// TwinCAT 3 PLC project TcAbbLinkin
// Title: TcAbbLinkin
// Company: Loupe
// Author: Loupe
// ProjectVersion: 0.1.0
// ProgramVersion: 3.1.4024.0
// libraries:
//   Tc2_Standard, * (Beckhoff Automation GmbH)
//   Tc2_System, * (Beckhoff Automation GmbH)
//   Tc2_Utilities, * (Beckhoff Automation GmbH)
//   Tc3_IotBase, * (Beckhoff Automation GmbH)
//   Tc3_JsonXml, * (Beckhoff Automation GmbH)
//   Tc3_Module, * (Beckhoff Automation GmbH)
// project tree:
//   DUTs/ AbbLinkinAuthDigest_Typ.TcDUT (not stored), AbbLinkinConfiguration_Typ.TcDUT, AbbLinkinRequestResults_Typ.TcDUT, AbbLinkinRequest_Typ.TcDUT (not stored), AbbLinkinRequestQueue_Typ.TcDUT (not stored), AbbLinkinRequestStatus_Typ.TcDUT, AbbLinkinAuth_Typ.TcDUT (not stored), ABBLINKIN_AUTH_HEADER_VALUE.TcDUT, ABBLINKIN_RWS_API_VERSION.TcDUT, ABBLINKIN_STATE.TcDUT, ABBLINKIN_COMMAND_TYPE.TcDUT, ABBLINKIN_DATA_TYPE_Typ.TcDUT (not stored), ABBLINKIN_STRING_EX_LEN.TcDUT
//   / PlcTask.TcTTO (not stored)
//   POUs/ MAIN.TcPOU, Example.TcPOU, TcAbbLinkin.TcPOU (not stored)
// real-time tasks:
//   TASK PlcTask: cycle T#10ms, priority 20, ADS port 350

// ---- DUTs/AbbLinkinConfiguration_Typ.TcDUT
// Copyright (c) 2024 Loupe (https://loupe.team), provided under the MIT License.
TYPE AbbLinkinConfiguration_Typ :
STRUCT
	rwsIpAddress : STRING := '127.0.0.1';
	rwsTcpPort : USINT := 80;
	rwsVersion : ABBLINKIN_RWS_API_VERSION;
	rwsUsername : STRING := 'Default User';
	rwsPassword : STRING := 'robotics';
	tlsAllowRwsCertSelfSigned : BOOL := FALSE;
	tlsCAFile : STRING(255) := '';
END_STRUCT
END_TYPE

// ---- DUTs/AbbLinkinRequestResults_Typ.TcDUT
// Copyright (c) 2024 Loupe (https://loupe.team), provided under the MIT License.
TYPE AbbLinkinRequestResults_Typ :
STRUCT
	pDataBool : POINTER TO BOOL;
	pDataDint : POINTER TO DINT;
	pDataLreal : POINTER TO LREAL;
	pDataString : POINTER TO STRING;
	dataType : ABBLINKIN_DATA_TYPE_Typ;
	dataLen : INT;
END_STRUCT
END_TYPE

// ---- DUTs/AbbLinkinRequestStatus_Typ.TcDUT
// Copyright (c) 2024 Loupe (https://loupe.team), provided under the MIT License.
TYPE AbbLinkinRequestStatus_Typ :
STRUCT
	busy : BOOL;
	done : BOOL;
	error : BOOL;
	errorID : DINT;
	errorMsg : STRING;
END_STRUCT
END_TYPE

// ---- DUTs/ABBLINKIN_AUTH_HEADER_VALUE.TcDUT
// Copyright (c) 2024 Loupe (https://loupe.team), provided under the MIT License.
{attribute 'qualified_only'}
{attribute 'strict'}
TYPE ABBLINKIN_AUTH_HEADER_VALUE :
(
	NONE,
	BASIC,
	DIGEST
);
END_TYPE

// ---- DUTs/ABBLINKIN_RWS_API_VERSION.TcDUT
// Copyright (c) 2024 Loupe (https://loupe.team), provided under the MIT License.
{attribute 'qualified_only'}
{attribute 'strict'}
TYPE ABBLINKIN_RWS_API_VERSION :
(
	V1 := 0,
	V2 := 2
);
END_TYPE

// ---- DUTs/ABBLINKIN_STATE.TcDUT
// Copyright (c) 2024 Loupe (https://loupe.team), provided under the MIT License.
{attribute 'qualified_only'}
{attribute 'strict'}
TYPE ABBLINKIN_STATE :
(
	IDLE,
	SEND_REQUEST,
	WAIT_FOR_RESONSE,
	PROCESS_RESPONSE,
	AUTH_START,
	AUTH_SEND_REQUEST,
	AUTH_WAIT_FOR_RESONSE,
	AUTH_PROCESS_RESPONSE,
	AUTH_DIGEST_RESPONSE_CALCULATE,
	AUTH_DIGEST_RESPONSE_SEND,
	ERROR
);
END_TYPE

// ---- DUTs/ABBLINKIN_COMMAND_TYPE.TcDUT
// Copyright (c) 2024 Loupe (https://loupe.team), provided under the MIT License.
{attribute 'qualified_only'}
{attribute 'strict'}
TYPE ABBLINKIN_COMMAND_TYPE :
(
	GET_IO,
	GET_CTRL_STATE,
	GET_OP_MODE,
	GET_RAPID_STATE,
	GET_SYMBOL,
	POWER_OFF,
	POWER_ON,
	RAPID_RESET,
	RAPID_START,
	RAPID_STOP,
	SET_IO,
	SET_SYMBOL
);
END_TYPE

// ---- DUTs/ABBLINKIN_STRING_EX_LEN.TcDUT
// Copyright (c) 2024 Loupe (https://loupe.team), provided under the MIT License.
TYPE ABBLINKIN_STRING_EX_LEN : STRING(2000); END_TYPE

// ---- POUs/MAIN.TcPOU
// Copyright (c) 2024 Loupe (https://loupe.team), provided under the MIT License.
PROGRAM MAIN
VAR
	myRobotLink : TcAbbLinkin;
	userSetConfigurationNow : BOOL := TRUE;
	userConnectStartNow : BOOL := TRUE;
	userConnectStopNow : BOOL;
	
	userGetCtrlStateNow : BOOL;
	userGetCtrlStateStatus : AbbLinkinRequestStatus_Typ;
	userGetCtrlStateResult : STRING;
	
	userGetOpModeNow : BOOL;
	userGetOpModeStatus : AbbLinkinRequestStatus_Typ;
	userGetOpModeResult : STRING;
	
	userGetRapidStateNow : BOOL;
	userGetRapidStateStatus : AbbLinkinRequestStatus_Typ;
	userGetRapidStateResult : STRING;
	
	userGetIoBoolNow : BOOL;
	userGetIoBoolStatus : AbbLinkinRequestStatus_Typ;
	userGetIoBoolResult : BOOL;
	
	userGetIoLrealNow : BOOL;
	userGetIoLrealStatus : AbbLinkinRequestStatus_Typ;
	userGetIoLrealResult : LREAL;
	
	userGetIoDintNow : BOOL;
	userGetIoDintStatus : AbbLinkinRequestStatus_Typ;
	userGetIoDintResult : DINT;
	
	
	userSetIoBoolNow : BOOL;
	userSetIoBoolValue : BOOL := 1;
	userSetIoBoolStatus : AbbLinkinRequestStatus_Typ;
	userSetIoDintNow : BOOL;
	userSetIoDintValue : DINT := 57;
	userSetIoDintStatus : AbbLinkinRequestStatus_Typ;
	userSetIoLrealNow : BOOL;
	userSetIoLrealValue : LREAL := 41.123456;
	userSetIoLrealStatus : AbbLinkinRequestStatus_Typ;
	
	
	userGetSymbolBoolNow : BOOL;
	userGetSymbolBoolResult : BOOL;
	userGetSymbolBoolStatus : AbbLinkinRequestStatus_Typ;
	userGetSymbolNumNow : BOOL;
	userGetSymbolNumResult : LREAL;
	userGetSymbolNumStatus : AbbLinkinRequestStatus_Typ;
	userGetSymbolStringNow : BOOL;
	userGetSymbolStringResult : STRING;
	userGetSymbolStringStatus : AbbLinkinRequestStatus_Typ;
	
	userSetSymbolBoolNow : BOOL;
	userSetSymbolBoolValue : BOOL := 1;
	userSetSymbolBoolStatus : AbbLinkinRequestStatus_Typ;
	userSetSymbolDintNow : BOOL;
	userSetSymbolDintValue : DINT := -57;
	userSetSymbolDintStatus : AbbLinkinRequestStatus_Typ;
	userSetSymbolLrealNow : BOOL;
	userSetSymbolLrealValue : LREAL := -41.123456;
	userSetSymbolLrealStatus : AbbLinkinRequestStatus_Typ;
	userSetSymbolStringNow : BOOL;
	userSetSymbolStringValue : STRING := 'test String';
	userSetSymbolStringStatus : AbbLinkinRequestStatus_Typ;
	userSetSymbolWStringNow : BOOL;
	userSetSymbolWStringValue : WSTRING := "test WString";
	userSetSymbolWStringStatus : AbbLinkinRequestStatus_Typ;
	
	
	userPowerOffNow : BOOL;
	userPowerOffStatus : AbbLinkinRequestStatus_Typ;
	userPowerOnNow : BOOL;
	userPowerOnStatus : AbbLinkinRequestStatus_Typ;
	userRapidResetNow : BOOL;
	userRapidResetStatus : AbbLinkinRequestStatus_Typ;
	userRapidStopNow : BOOL;
	userRapidStopStatus : AbbLinkinRequestStatus_Typ;
	userRapidStartNow : BOOL;
	userRapidStartStatus : AbbLinkinRequestStatus_Typ;
	
	
	userAckErrorNow : BOOL;
END_VAR

// Set configuration
if userSetConfigurationNow then
	myRobotLink.configuration.rwsIpAddress := '127.0.0.1';
	myRobotLink.configuration.rwsTcpPort := 80;
	myRobotLink.configuration.rwsVersion := ABBLINKIN_RWS_API_VERSION.V2;
	myRobotLink.configuration.rwsUsername := 'Default User';
	myRobotLink.configuration.rwsPassword := 'robotics';
	//myRobotLink.configuration.tlsAllowRwsCertSelfSigned := TRUE;
	myRobotLink.configuration.tlsAllowRwsCertSelfSigned := FALSE;
	myRobotLink.configuration.tlsCAFile := 'C:\TwinCAT\3.1\Config\Certificates\TcAbbLinkinCA.pem';
	
	userSetConfigurationNow := FALSE;
END_IF


// Cyclic
myRobotLink.Cyclic();


IF userConnectStartNow THEN
	myRobotLink.Connect();
	userConnectStartNow := FALSE;
END_IF

IF userConnectStopNow THEN
	myRobotLink.Disconnect();
	userConnectStopNow := FALSE;
END_IF


IF userGetCtrlStateNow THEN
	myRobotLink.GetCtrlState(ADR(userGetCtrlStateStatus), ADR(userGetCtrlStateResult));
	userGetCtrlStateNow := FALSE;
END_IF


IF userGetOpModeNow THEN
	myRobotLink.GetOpMode(ADR(userGetOpModeStatus), ADR(userGetOpModeResult));
	userGetOpModeNow := FALSE;
END_IF


IF userGetRapidStateNow THEN
	myRobotLink.GetRapidState(ADR(userGetRapidStateStatus), ADR(userGetRapidStateResult));
	userGetRapidStateNow := FALSE;
END_IF


IF userGetIoBoolNow THEN
	myRobotLink.GetIODigital(signal := 'myInputDIG', pStatus := ADR(userGetIoBoolStatus), pResult := ADR(userGetIoBoolResult));
	userGetIoBoolNow := FALSE;
END_IF

IF userGetIoLrealNow THEN
	myRobotLink.GetIOAnalog(signal := 'myInputANA', pStatus := ADR(userGetIoLrealStatus), pResult := ADR(userGetIoLrealResult));
	userGetIoLrealNow := FALSE;
END_IF

IF userGetIoDintNow THEN
	myRobotLink.GetIOGroup(signal := 'myInputGRP', pStatus := ADR(userGetIoDintStatus), pResult := ADR(userGetIoDintResult));
	userGetIoDintNow := FALSE;
END_IF


IF userSetIoBoolNow THEN
	myRobotLink.SetIO('myInputDIG', userSetIoBoolValue, ADR(userSetIoBoolStatus));
	userSetIoBoolNow := FALSE;
END_IF
IF userSetIoDintNow THEN
	myRobotLink.SetIO('myInputGRP', userSetIoDintValue, ADR(userSetIoDintStatus));
	userSetIoDintNow := FALSE;
END_IF
IF userSetIoLrealNow THEN
	myRobotLink.SetIO('myInputANA', userSetIoLrealValue, ADR(userSetIoLrealStatus));
	userSetIoLrealNow := FALSE;
END_IF


IF userGetSymbolBoolNow THEN
	myRobotLink.GetSymbolBool(symbolUrl := 'RAPID/T_ROB1/Module1/myRapidBool', pStatus := ADR(userGetSymbolBoolStatus), pResult := ADR(userGetSymbolBoolResult));
	userGetSymbolBoolNow := FALSE;
END_IF
IF userGetSymbolNumNow THEN
	myRobotLink.GetSymbolNum(symbolUrl := 'RAPID/T_ROB1/Module1/myRapidNum', pStatus := ADR(userGetSymbolNumStatus), pResult := ADR(userGetSymbolNumResult));
	userGetSymbolNumNow := FALSE;
END_IF
IF userGetSymbolStringNow THEN
	myRobotLink.GetSymbolString(symbolUrl := 'RAPID/T_ROB1/Module1/myRapidString', pStatus := ADR(userGetSymbolStringStatus), pResult := ADR(userGetSymbolStringResult));
	userGetSymbolStringNow := FALSE;
END_IF


IF userSetSymbolBoolNow THEN
	myRobotLink.SetSymbol('RAPID/T_ROB1/Module1/myRapidBool', userSetSymbolBoolValue, ADR(userSetSymbolBoolStatus));
	userSetSymbolBoolNow := FALSE;
END_IF
IF userSetSymbolDintNow THEN
	myRobotLink.SetSymbol('RAPID/T_ROB1/Module1/myRapidNum', userSetSymbolDintValue, ADR(userSetSymbolDintStatus));
	userSetSymbolDintNow := FALSE;
END_IF
IF userSetSymbolLrealNow THEN
	myRobotLink.SetSymbol('RAPID/T_ROB1/Module1/myRapidNum', userSetSymbolLrealValue, ADR(userSetSymbolLrealStatus));
	userSetSymbolLrealNow := FALSE;
END_IF
IF userSetSymbolStringNow THEN
	myRobotLink.SetSymbol('RAPID/T_ROB1/Module1/myRapidString', userSetSymbolStringValue, ADR(userSetSymbolStringStatus));
	userSetSymbolStringNow := FALSE;
END_IF
IF userSetSymbolWStringNow THEN
	myRobotLink.SetSymbol('RAPID/T_ROB1/Module1/myRapidString', userSetSymbolWStringValue, ADR(userSetSymbolWStringStatus));
	userSetSymbolWStringNow := FALSE;
END_IF


IF userPowerOffNow THEN
	myRobotLink.PowerOff(ADR(userPowerOffStatus));
	userPowerOffNow := FALSE;
END_IF
IF userPowerOnNow THEN
	myRobotLink.PowerOn(ADR(userPowerOnStatus));
	userPowerOnNow := FALSE;
END_IF
IF userRapidResetNow THEN
	myRobotLink.RapidReset(ADR(userRapidResetStatus));
	userRapidResetNow := FALSE;
END_IF
IF userRapidStopNow THEN
	myRobotLink.RapidStop(ADR(userRapidStopStatus));
	userRapidStopNow := FALSE;
END_IF
IF userRapidStartNow THEN
	myRobotLink.RapidStart(ADR(userRapidStartStatus));
	userRapidStartNow := FALSE;
END_IF


IF userAckErrorNow THEN
	myRobotLink.AckError();
	userAckErrorNow := FALSE;
END_IF

END_PROGRAM

// ---- POUs/Example.TcPOU
// Copyright (c) 2024 Loupe (https://loupe.team), provided under the MIT License.
PROGRAM Example
VAR
	myRobotLink : TcAbbLinkin;
	initConfiguration : BOOL := TRUE;
	initConnection : BOOL := TRUE;
	userCommand_GetCtrlState : BOOL := TRUE;
	getCtrlStateStatus : AbbLinkinRequestStatus_Typ;
	currentState : STRING;
	output : STRING;
END_VAR

// Initialize configuration
IF initConfiguration THEN
	myRobotLink.configuration.rwsIpAddress := '127.0.0.1';
	myRobotLink.configuration.rwsTcpPort := 80;
	myRobotLink.configuration.rwsVersion := ABBLINKIN_RWS_API_VERSION.V2;
	myRobotLink.configuration.rwsUsername := 'Default User';
	myRobotLink.configuration.rwsPassword := 'robotics';
	myRobotLink.configuration.tlsAllowRwsCertSelfSigned := TRUE;
	
	initConfiguration := FALSE;
END_IF

myRobotLink.Cyclic();

/////////////////////////
// Connect
IF initConnection THEN
	myRobotLink.Connect();
	initConnection := FALSE;
END_IF

/////////////////////////
// Get State

// Send command
IF myRobotLink.readyForCmd AND userCommand_GetCtrlState THEN
	myRobotLink.GetCtrlState(pStatus := ADR(getCtrlStateStatus), pResultState := ADR(currentState));
	userCommand_GetCtrlState := FALSE;
END_IF

// Process Results
IF getCtrlStateStatus.done THEN
	output := CONCAT('Current state is ', currentState);
ELSIF getCtrlStateStatus.error THEN
	output := 'An Error occured.';
END_IF

END_PROGRAM
